SYSTEM IWORFRAUD (* System Configuration *)
  (* Standard: 61499-1 *)
  (* Version 0.3, 2003-12-05, JHC, Rockwell Automation, Renamed from NEWSYSTEM. *)
  (* Version 0.2, 2002-11-05, JHC, Rockwell Automation, Fixed missing (empty) FBD in Application. *)
  (* Version 0.1, 2002-01-17, JHC, Rockwell Automation, Minor cleanup *)
  (* Version 0.0, 2000-05-27, JHC, Rockwell Automation *)
  APPLICATION APP1
  END_APPLICATION
  DEVICE Controller : FRAME_DEVICE
    RESOURCE RES1 : PANEL_RESOURCE
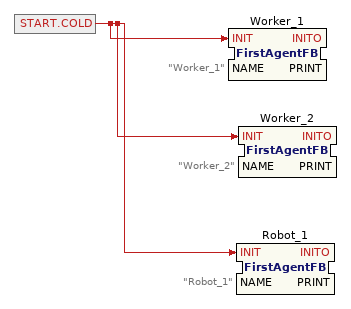
      FBS
        Worker_1 : FirstAgentFB(NAME := "Worker_1");
        Worker_2 : FirstAgentFB(NAME := "Worker_2");
        Robot_1 : FirstAgentFB(NAME := "Robot_1");
      END_FBS
      EVENT_CONNECTIONS
        START.COLD TO Worker_1.INIT;
        START.COLD TO Worker_2.INIT;
        START.COLD TO Robot_1.INIT;
      END_CONNECTIONS
    END_RESOURCE
  END_DEVICE
END_SYSTEM
